{attribute 'linkalways'} 
{attribute 'no_explicit_call' := 'This FB is a CLASS and must be accessed using methods or properties'}
{attribute 'enable_dynamic_creation'}
FUNCTION_BLOCK ABSTRACT Alarm IMPLEMENTS I_Alarm

METHOD PUBLIC Accept
VAR_INPUT
	Visitor : I_AlarmVisitor;
END_VAR
Visitor.VisitAlarm(THIS^);
END_METHOD

PROPERTY ABSTRACT Active : BOOL
GET
END_GET
END_PROPERTY

METHOD ABSTRACT Clear
END_METHOD

METHOD FB_init : BOOL
VAR_INPUT
	bInitRetains : BOOL; // if TRUE, the retain variables are initialized (warm start / cold start)
	bInCopyCode : BOOL;  // if TRUE, the instance afterwards gets moved into the copy code (online change)
	Parent : I_HostAlarms;
END_VAR
RegisterWithParent(Parent);
END_METHOD

PROPERTY ABSTRACT Message : T_MaxString
GET
END_GET
END_PROPERTY

PROPERTY ABSTRACT Reason : T_MaxString
GET
END_GET
END_PROPERTY

METHOD RegisterWithParent
VAR_INPUT
	Parent : I_HostAlarms;
END_VAR
IF Parent = 0 THEN
	RETURN;
END_IF

Parent.Alarms.AddAlarm(THIS^);
END_METHOD

METHOD PUBLIC SerializeWith
VAR_INPUT
	Serializer : I_Serializer;
END_VAR
VAR
	isActive : BOOL := Active;
	errorMessage : T_MAXSTRING := Message;
	reasonMessage : T_MAXSTRING := Reason;
END_VAR
Serializer.StartObject();
Serializer.AddKeyString('message', errorMessage);
Serializer.AddKeyBool('active', isActive);

IF reasonMessage <> '' THEN
	Serializer.AddKeyString('reason', reasonMessage);
END_IF

Serializer.EndObject();
END_METHOD

END_FUNCTION_BLOCK

(* stored: Version 1.1.0.1, ProductVersion 3.1.4024.13
   POU Alarm: Id {dc64a02b-06d6-4cd6-bb49-ecdb4c808ffc}, SpecialFunc None
   Folder Abstract: Id {5c2dccff-8f73-4f38-99b0-0f34aeffa2e8}
   Folder Constructor: Id {04ae702e-640d-4d81-b27b-89d8b86cec46}
   Method Accept: Id {cb96dbd8-c488-49a7-8481-6535755fd321}
   Property Active: Id {b38435b1-3786-40d3-9015-61a5a18fb496}
   Get Get: Id {db4f51d3-ea95-4356-b237-909d78d4cf9c}
   Method Clear: Id {4b1d35fc-269d-4478-9303-7ca63493254d}
   Method FB_init: Id {c56eac3a-81df-4abd-83f3-880c190ff443}
   Property Message: Id {0fbccf42-8732-44ef-b561-8de47087a052}
   Get Get: Id {fe52d97c-2162-4120-ba0d-42aa6ff7b326}
   Property Reason: Id {1e9d7ed8-a7d6-4aa9-9157-c12bfbfb87f2}
   Get Get: Id {f38c9c34-4550-4d70-8e00-5fd8be5615ea}
   Method RegisterWithParent: Id {8717cda6-ea38-404c-9eb7-e5632b2f7e4f}
   Method SerializeWith: Id {2d3a51b2-3b6b-44a7-b71a-926f8c47e140} *)
